# B&R Automation Studio project reAM250plc (part 8)

#### CustomStatemachineRecoater.cpp
```cpp
/*++

Copyright (C) 2024 Institute for Machine Tools and Industrial Management
TUM School of Engineering and Design
Technical University of Munich

All rights reserved.

Redistribution and use in source and binary forms, with or without
modification, are permitted provided that the following conditions are met:
	* Redistributions of source code must retain the above copyright
	  notice, this list of conditions and the following disclaimer.
	* Redistributions in binary form must reproduce the above copyright
	  notice, this list of conditions and the following disclaimer in the
	  documentation and/or other materials provided with the distribution.
	* Neither the name of the Technical University of Munich nor the
	  names of its contributors may be used to endorse or promote products
	  derived from this software without specific prior written permission.

THIS SOFTWARE IS PROVIDED BY THE COPYRIGHT HOLDERS AND CONTRIBUTORS "AS IS" AND
ANY EXPRESS OR IMPLIED WARRANTIES, INCLUDING, BUT NOT LIMITED TO, THE IMPLIED
WARRANTIES OF MERCHANTABILITY AND FITNESS FOR A PARTICULAR PURPOSE ARE
DISCLAIMED. IN NO EVENT SHALL TECHNICAL UNIVERSITY OF MUNICH BE LIABLE FOR ANY
DIRECT, INDIRECT, INCIDENTAL, SPECIAL, EXEMPLARY, OR CONSEQUENTIAL DAMAGES
(INCLUDING, BUT NOT LIMITED TO, PROCUREMENT OF SUBSTITUTE GOODS OR SERVICES;
LOSS OF USE, DATA, OR PROFITS; OR BUSINESS INTERRUPTION) HOWEVER CAUSED AND
ON ANY THEORY OF LIABILITY, WHETHER IN CONTRACT, STRICT LIABILITY, OR TORT
(INCLUDING NEGLIGENCE OR OTHERWISE) ARISING IN ANY WAY OUT OF THE USE OF THIS
SOFTWARE, EVEN IF ADVISED OF THE POSSIBILITY OF SUCH DAMAGE.

*/

#include "Framework/Application.hpp"

#include "CustomConstants.hpp"

//include required hardware modules
#include "Modules/IOModule_X20DO6322.hpp"
#include "Modules/IOModule_X20DI6371.hpp"
#include "Modules/MappMotion_SingleAxis.hpp"
#include "Modules/IOModule_X20SC0842.hpp"

namespace BuRCPP {

	class CStateRecoaterAxes_WaitForInit : public CState {
		public:

		std::string getName ()
		{
			return "wait_for_init";
		}

		void Execute (CEnvironment * pEnvironment)
		{
			pEnvironment->setNextState("wait_for_init");
			// access an IO modules
			ioModuleAccess<CMappMotion_SingleLinearAxis> pRecoaterAxisLinearModule (pEnvironment, "RecoaterLinear");
			ioModuleAccess<CMappMotion_SingleLinearAxis> pRecoaterAxisPowderbeltModule (pEnvironment, "RecoaterAxisPowderbelt");

			// check for PC signals
			auto pSignalInitRecoateraxisPowder = pEnvironment->checkSignal ("initpowderaxis");
			auto pSignalInitRecoateraxisLinear = pEnvironment->checkSignal ("initlinearaxis");

			// get journal variables
			auto bInitRecoateraxisPowder = pEnvironment->getBoolValue(JOURNALVARIABLE_INITRECOATERPOWDERBELT);
			auto bInitRecoateraxisLinear = pEnvironment->getBoolValue(JOURNALVARIABLE_INITRECOATERLINEAR);

			if(bInitRecoateraxisPowder && bInitRecoateraxisLinear)
			{
				// wait for PC signal to init
				pEnvironment->setNextState("init");
			}
			else if(pSignalInitRecoateraxisPowder)
			{
				pEnvironment->setBoolValue(JOURNALVARIABLE_INITRECOATERPOWDERBELT, true);
				pSignalInitRecoateraxisPowder->setBoolResult("success", true);
				pSignalInitRecoateraxisPowder->finishProcessing ();
			}
			else if (pSignalInitRecoateraxisLinear)
			{
				pEnvironment->setBoolValue(JOURNALVARIABLE_INITRECOATERLINEAR, true);
				pSignalInitRecoateraxisLinear->setBoolResult("success", true);
				pSignalInitRecoateraxisLinear->finishProcessing ();
			}
			else if (pRecoaterAxisLinearModule-> isError () || pRecoaterAxisPowderbeltModule-> isError ())
			{
				pEnvironment->setNextState ("error");
			}
			else
			{
				pEnvironment->setNextState("wait_for_init");
			}

		}
	};

	class CStateRecoaterAxes_Init : public CState {
		public:

		std::string getName ()
		{
			return "init";
		}

		void Execute (CEnvironment * pEnvironment)
		{
			// access an IO modules
			ioModuleAccess<CMappMotion_SingleLinearAxis> pRecoaterAxisLinearModule (pEnvironment, "RecoaterLinear");
			ioModuleAccess<CMappMotion_SingleLinearAxis> pRecoaterAxisPowderbeltModule (pEnvironment, "RecoaterAxisPowderbelt");

			if (pRecoaterAxisLinearModule->canSetPower () && pRecoaterAxisPowderbeltModule->canSetPower () )
			{
				if(pRecoaterAxisLinearModule->isReferenced () && pRecoaterAxisLinearModule->isReferenced ())
				{
					pRecoaterAxisLinearModule->setPower(true);
					pRecoaterAxisPowderbeltModule->setPower(true);
					pEnvironment->setNextState ("idle");
				}
				else
				{
					pRecoaterAxisLinearModule->setPowerOnAndStartReference ();
					pRecoaterAxisPowderbeltModule->setPowerOnAndStartReference ();
					pEnvironment->setNextState ("wait_for_referencing");
				}

			}
			else if (pRecoaterAxisLinearModule-> isError () || pRecoaterAxisPowderbeltModule-> isError ())
			{
				pEnvironment->setNextState ("error");
			}
			else
			{
				pEnvironment->setNextState ("init");
			}

		}
	};

	class CStateRecoaterAxes_Idle : public CState {
		public:

		std::string getName ()
		{
			return "idle";
		}

		void Execute (CEnvironment * pEnvironment)
		{
			pEnvironment->setNextState("idle");

			// access an IO modules
			ioModuleAccess<CMappMotion_SingleLinearAxis> pRecoaterAxisLinearModule (pEnvironment, "RecoaterLinear");
			ioModuleAccess<CMappMotion_SingleLinearAxis> pRecoaterAxisPowderbeltModule (pEnvironment, "RecoaterAxisPowderbelt");

			// check for PC signals
			auto pSignalReferenceAxis = pEnvironment->checkSignal ("referenceaxis");
			auto pSignalSingleAxisMovement = pEnvironment->checkSignal ("triggersingleaxismovement");
			auto pSignalDualAxisMovement = pEnvironment->checkSignal ("recoaterdualaxismovement");

			if (pSignalReferenceAxis)
			{
				bool referenceRecoaterAxisLinear = pSignalReferenceAxis->getBoolParameter("reference_recoateraxis_linear");
				bool referenceRecoaterAxisPowder = pSignalReferenceAxis->getBoolParameter("reference_recoateraxis_powder");

				if (referenceRecoaterAxisLinear || referenceRecoaterAxisLinear)
				{
					pEnvironment->setIntegerValue(JOURNALVARIABLE_REFERENCERECOATERPOWDERBELT, referenceRecoaterAxisPowder);
					pEnvironment->setIntegerValue(JOURNALVARIABLE_REFERENCERECOATERLINEAR, referenceRecoaterAxisLinear);
					pEnvironment->setNextState("manual_referencing");
					pSignalReferenceAxis->finishProcessing ();
					return;
				}
			}
			if (pSignalSingleAxisMovement)
			{
				int axisid = pSignalSingleAxisMovement->getInt32Parameter("axisid");
				if (axisid == AXISID_RECOATELINEAR)
				{
					pEnvironment->setNextState("linear_axis_movement");
					pEnvironment->setIntegerValue(JOURNALVARIABLE_RECOATERLINEARMOVEMENTABSOLUTERELATIVE, pSignalSingleAxisMovement->getInt32Parameter("absoluterelative"));
					pEnvironment->setDoubleValue(JOURNALVARIABLE_RECOATERLINEARMOVEMENTPOSITION, pSignalSingleAxisMovement->getInt32Parameter("position") * 0.001);
					pEnvironment->setDoubleValue(JOURNALVARIABLE_RECOATERLINEARMOVEMENTSPEED, pSignalSingleAxisMovement->getInt32Parameter("speed") * 0.001);
					pEnvironment->setDoubleValue(JOURNALVARIABLE_RECOATERLINEARMOVEMENTACCELERATION, pSignalSingleAxisMovement->getInt32Parameter("acceleration") * 0.001);
					pSignalSingleAxisMovement->finishProcessing ();
					return;
				}
				else if (axisid == AXISID_RECOATERPOWDERBELT)
				{
					pEnvironment->setNextState("powder_belt_axis_movement");
					pEnvironment->setIntegerValue(JOURNALVARIABLE_RECOATERPOWDERBELTMOVEMENTABSOLUTERELATIVE, pSignalSingleAxisMovement->getInt32Parameter("absoluterelative"));
					pEnvironment->setDoubleValue(JOURNALVARIABLE_RECOATERPOWDERBELTMOVEMENTPOSITION, pSignalSingleAxisMovement->getInt32Parameter("position") * 0.001);
					pEnvironment->setDoubleValue(JOURNALVARIABLE_RECOATERPOWDERBELTMOVEMENTSPEED, pSignalSingleAxisMovement->getInt32Parameter("speed") * 0.001);
					pEnvironment->setDoubleValue(JOURNALVARIABLE_RECOATERPOWDERBELTMOVEMENTACCELERATION, pSignalSingleAxisMovement->getInt32Parameter("acceleration") * 0.001);
					pSignalSingleAxisMovement->finishProcessing ();
					return;
				}
			}
			if (pSignalDualAxisMovement)
			{
				pEnvironment->setNextState("dual_axis_movement");
				pEnvironment->setDoubleValue(JOURNALVARIABLE_RECOATERMOVEMENTSTARTPOSITION, pSignalDualAxisMovement->getInt32Parameter("recoateraxis_linear_start_position") * 0.001);
				pEnvironment->setDoubleValue(JOURNALVARIABLE_RECOATERMOVEMENTTARGETPOSITION, pSignalDualAxisMovement->getInt32Parameter("recoateraxis_linear_target_position") * 0.001);
				pEnvironment->setDoubleValue(JOURNALVARIABLE_RECOATERMOVEMENTLINEARAXISSPEED, pSignalDualAxisMovement->getInt32Parameter("recoateraxis_linear_speed") * 0.001);
				pEnvironment->setDoubleValue(JOURNALVARIABLE_RECOATERMOVEMENTPOWDERAXISSPEED, pSignalDualAxisMovement->getInt32Parameter("recoateraxis_powder_speed") * 0.001);
				pEnvironment->setDoubleValue(JOURNALVARIABLE_RECOATERMOVEMENTLINEARAXISACCELERATION, pSignalDualAxisMovement->getInt32Parameter("recoater_axes_linear_acceleration") * 0.001);
				pEnvironment->setDoubleValue(JOURNALVARIABLE_RECOATERMOVEMENTPOWDERAXISACCELERATION, pSignalDualAxisMovement->getInt32Parameter("recoater_axes_powder_acceleration") * 0.001);
				pSignalDualAxisMovement->finishProcessing ();
			}
			if (pRecoaterAxisLinearModule-> isError () || pRecoaterAxisPowderbeltModule-> isError ())
			{
				pEnvironment->setNextState ("error");
			}
		}
	};

	class CStateRecoaterAxes_LinearAxisMovement : public CState {
		public:

		std::string getName ()
		{
			return "linear_axis_movement";
		}

		void Execute (CEnvironment * pEnvironment)
		{
			pEnvironment->setNextState("linear_axis_movement");

			// access an IO modules
			ioModuleAccess<CMappMotion_SingleLinearAxis> pRecoaterAxisLinearModule (pEnvironment, "RecoaterLinear");

			if (pRecoaterAxisLinearModule->canMoveAxis ())
			{
				auto absoluterelative = pEnvironment->getInt32Value(JOURNALVARIABLE_RECOATERLINEARMOVEMENTABSOLUTERELATIVE);
				auto position = pEnvironment->getDoubleValue(JOURNALVARIABLE_RECOATERLINEARMOVEMENTPOSITION);
				auto speed = pEnvironment->getDoubleValue(JOURNALVARIABLE_RECOATERLINEARMOVEMENTSPEED);
				auto acceleration = pEnvironment->getDoubleValue(JOURNALVARIABLE_RECOATERLINEARMOVEMENTACCELERATION);

				if (absoluterelative == AXISMOVEMENT_ABSOLUTE){
					pRecoaterAxisLinearModule->moveAxisAbsolute (position, speed, acceleration);

				}else if (absoluterelative == AXISMOVEMENT_RELATIVE){
					pRecoaterAxisLinearModule->moveAxisRelative (position, speed, acceleration);
				}
				pEnvironment->setNextState ("wait_for_linear_axis_movement");
			}
			else if (pRecoaterAxisLinearModule-> isError ())
			{
				pEnvironment->setNextState ("error");
			}
			else
			{
				pEnvironment->setNextState ("linear_axis_movement");
			}
		}

	};

	class CStateRecoaterAxes_WaitForLinearAxisMovement : public CState {
		public:

		std::string getName ()
		{
			return "wait_for_linear_axis_movement";
		}

		void Execute (CEnvironment * pEnvironment)
		{
			pEnvironment->setNextState("wait_for_linear_axis_movement");

			// access an IO modules
			ioModuleAccess<CMappMotion_SingleLinearAxis> pRecoaterAxisLinearModule (pEnvironment, "RecoaterLinear");

			if (pRecoaterAxisLinearModule->isInPosition())
			{
				pEnvironment->setNextState ("idle");
			}
			else if (pRecoaterAxisLinearModule-> isError ())
			{
				pEnvironment->setNextState ("error");
			}
			else
			{
				pEnvironment->setNextState ("wait_for_linear_axis_movement");
			}

		}

	};

	class CStateRecoaterAxes_PowderBeltAxisMovement : public CState {
		public:

		std::string getName ()
		{
			return "powder_belt_axis_movement";
		}

		void Execute (CEnvironment * pEnvironment)
		{
			pEnvironment->setNextState("powder_belt_axis_movement");

			// access an IO modules
			ioModuleAccess<CMappMotion_SingleLinearAxis> pRecoaterAxisPowderbeltModule (pEnvironment, "RecoaterAxisPowderbelt");

			if (pRecoaterAxisPowderbeltModule->canMoveAxis ())
			{
				auto absoluterelative = pEnvironment->getInt32Value(JOURNALVARIABLE_RECOATERPOWDERBELTMOVEMENTABSOLUTERELATIVE);
				auto position = pEnvironment->getDoubleValue(JOURNALVARIABLE_RECOATERPOWDERBELTMOVEMENTPOSITION);
				auto speed = pEnvironment->getDoubleValue(JOURNALVARIABLE_RECOATERPOWDERBELTMOVEMENTSPEED);
				auto acceleration = pEnvironment->getDoubleValue(JOURNALVARIABLE_RECOATERPOWDERBELTMOVEMENTACCELERATION);

				if (absoluterelative == AXISMOVEMENT_ABSOLUTE){
					pRecoaterAxisPowderbeltModule->moveAxisAbsolute (position, speed, acceleration);

				}else if (absoluterelative == AXISMOVEMENT_RELATIVE){
					pRecoaterAxisPowderbeltModule->moveAxisRelative (position, speed, acceleration);
				}
				pEnvironment->setNextState ("wait_for_powder_belt_axis_movement");
			}
			else if (pRecoaterAxisPowderbeltModule-> isError ())
			{
				pEnvironment->setNextState ("error");
			}
			else
			{
				pEnvironment->setNextState ("powder_belt_axis_movement");
			}
		}

	};

	class CStateRecoaterAxes_WaitForPowderBeltAxisMovement : public CState {
		public:

		std::string getName ()
		{
			return "wait_for_powder_belt_axis_movement";
		}

		void Execute (CEnvironment * pEnvironment)
		{
			pEnvironment->setNextState("wait_for_powder_belt_axis_movement");

			// access an IO modules
			ioModuleAccess<CMappMotion_SingleLinearAxis> pRecoaterAxisPowderbeltModule (pEnvironment, "RecoaterAxisPowderbelt");

			if (pRecoaterAxisPowderbeltModule->isInPosition())
			{
				pEnvironment->setNextState ("idle");
			}
			else if (pRecoaterAxisPowderbeltModule-> isError ())
			{
				pEnvironment->setNextState ("error");
			}
			else
			{
				pEnvironment->setNextState ("wait_for_powder_belt_axis_movement");
			}

		}

	};

	class CStateRecoaterAxes_DualAxisMovement : public CState {
		public:

		std::string getName ()
		{
			return "dual_axis_movement";
		}

		void Execute (CEnvironment * pEnvironment)
		{
			pEnvironment->setNextState("dual_axis_movement");

			// access an IO modules
			ioModuleAccess<CMappMotion_SingleLinearAxis> pRecoaterAxisLinearModule (pEnvironment, "RecoaterLinear");
			ioModuleAccess<CMappMotion_SingleLinearAxis> pRecoaterAxisPowderbeltModule (pEnvironment, "RecoaterAxisPowderbelt");

			if (pRecoaterAxisLinearModule->canMoveAxis () && pRecoaterAxisPowderbeltModule->canMoveAxis ())
			{
				auto recoateraxis_linear_start_position = pEnvironment->getDoubleValue(JOURNALVARIABLE_RECOATERMOVEMENTSTARTPOSITION);
				auto recoateraxis_linear_target_position = pEnvironment->getDoubleValue(JOURNALVARIABLE_RECOATERMOVEMENTTARGETPOSITION);
				auto recoateraxis_linear_speed = pEnvironment->getDoubleValue(JOURNALVARIABLE_RECOATERMOVEMENTLINEARAXISSPEED);
				auto recoateraxis_powder_speed = pEnvironment->getDoubleValue(JOURNALVARIABLE_RECOATERMOVEMENTPOWDERAXISSPEED);
				auto recoater_axes_linear_acceleration = pEnvironment->getDoubleValue(JOURNALVARIABLE_RECOATERMOVEMENTLINEARAXISACCELERATION);
				auto recoater_axes_powder_acceleration = pEnvironment->getDoubleValue(JOURNALVARIABLE_RECOATERMOVEMENTPOWDERAXISACCELERATION);

				pRecoaterAxisLinearModule->moveAxisAbsolute (recoateraxis_linear_target_position, recoateraxis_linear_speed, recoater_axes_linear_acceleration);
				auto recoateraxis_powder_target_position = ((-(recoateraxis_linear_target_position-recoateraxis_linear_start_position))/recoateraxis_linear_speed)*recoateraxis_powder_speed;
				pRecoaterAxisPowderbeltModule->moveAxisRelative (recoateraxis_powder_target_position, recoateraxis_powder_speed, recoater_axes_powder_acceleration);

				pEnvironment->setNextState ("wait_for_dual_axis_movement");
			}
			else if (pRecoaterAxisLinearModule-> isError () || pRecoaterAxisPowderbeltModule-> isError ())
			{
				pEnvironment->setNextState ("error");
			}
			else
			{
				pEnvironment->setNextState ("dual_axis_movement");
			}
		}

	};

	class CStateRecoaterAxes_WaitForDualAxisMovement : public CState {
		public:

		std::string getName ()
		{
			return "wait_for_dual_axis_movement";
		}

		void Execute (CEnvironment * pEnvironment)
		{
			pEnvironment->setNextState("wait_for_dual_axis_movement");

			// access an IO modules
			ioModuleAccess<CMappMotion_SingleLinearAxis> pRecoaterAxisLinearModule (pEnvironment, "RecoaterLinear");
			ioModuleAccess<CMappMotion_SingleLinearAxis> pRecoaterAxisPowderbeltModule (pEnvironment, "RecoaterAxisPowderbelt");

			if (pRecoaterAxisLinearModule->isInPosition() && pRecoaterAxisPowderbeltModule->isInPosition())
			{
				pEnvironment->setNextState ("idle");
			}
			else if (pRecoaterAxisLinearModule-> isError () || pRecoaterAxisPowderbeltModule-> isError ())
			{
				pEnvironment->setNextState ("error");
			}
			else
			{
				pEnvironment->setNextState ("wait_for_dual_axis_movement");
			}

		}

	};

	class CStateRecoaterAxes_ManualReferencing : public CState {
		public:

		std::string getName ()
		{
			return "manual_referencing";
		}

		void Execute (CEnvironment * pEnvironment)
		{
			// access an IO modules
			ioModuleAccess<CMappMotion_SingleLinearAxis> pRecoaterAxisLinearModule (pEnvironment, "RecoaterLinear");
			ioModuleAccess<CMappMotion_SingleLinearAxis> pRecoaterAxisPowderbeltModule (pEnvironment, "RecoaterAxisPowderbelt");

			auto referenceRecoaterAxisLinear = pEnvironment->getInt32Value(JOURNALVARIABLE_REFERENCERECOATERLINEAR);
			auto referenceRecoaterAxisPowder = pEnvironment->getInt32Value(JOURNALVARIABLE_REFERENCERECOATERPOWDERBELT);

			if (pRecoaterAxisLinearModule-> isError () || pRecoaterAxisPowderbeltModule-> isError ())
			{
				pEnvironment->setNextState ("error");
			}
			else if (referenceRecoaterAxisLinear || referenceRecoaterAxisPowder)
			{
				if (referenceRecoaterAxisLinear)
				{
					pRecoaterAxisLinearModule->startReference ();
				}
				if (referenceRecoaterAxisPowder)
				{
					pRecoaterAxisPowderbeltModule->startReference ();
				}
				pEnvironment->setNextState("wait_for_referencing");
			}
			else
			{
				pEnvironment->setNextState("manual_referencing");
			}

		}

	};

	class CStateRecoaterAxes_WaitForReferencing : public CState {
		public:

		std::string getName ()
		{
			return "wait_for_referencing";
		}

		void Execute (CEnvironment * pEnvironment)
		{
			pEnvironment->setNextState("wait_for_referencing");

			// access an IO modules
			ioModuleAccess<CMappMotion_SingleLinearAxis> pRecoaterAxisLinearModule (pEnvironment, "RecoaterLinear");
			ioModuleAccess<CMappMotion_SingleLinearAxis> pRecoaterAxisPowderbeltModule (pEnvironment, "RecoaterAxisPowderbelt");

			if (pRecoaterAxisLinearModule-> isError () || pRecoaterAxisPowderbeltModule-> isError ())
			{
				pEnvironment->setNextState ("error");
			}
			else if(pRecoaterAxisLinearModule->isReferenced () && pRecoaterAxisPowderbeltModule->isReferenced ())
			{
				pEnvironment->setNextState("idle");
			}
			else
			{
				pEnvironment->setNextState("wait_for_referencing");
			}

		}

	};

	class CStateRecoaterAxes_Error : public CState {
		public:

		std::string getName ()
		{
			return "error";
		}

		void Execute (CEnvironment * pEnvironment)
		{
			pEnvironment->setNextState("error");

			// access an IO modules
			ioModuleAccess<CMappMotion_SingleLinearAxis> pRecoaterAxisLinearModule (pEnvironment, "RecoaterLinear");
			ioModuleAccess<CMappMotion_SingleLinearAxis> pRecoaterAxisPowderbeltModule (pEnvironment, "RecoaterAxisPowderbelt");
			ioModuleAccess<CIOModule_X20SC0842> pSafeDigitalInputModule115KF53 (pEnvironment, "115KF53"); //acknowledge button

			if(pSafeDigitalInputModule115KF53->getInput(2) == 1) //acknowledge button pressed
			{
				pRecoaterAxisLinearModule->resetError ();
				pRecoaterAxisPowderbeltModule->resetError ();
			}

			if (pRecoaterAxisLinearModule-> isError () || pRecoaterAxisPowderbeltModule-> isError ())
			{
				pEnvironment->setNextState ("error");
			}
			else
			{
				pEnvironment->setNextState ("init");
			}

		}

	};

	class CStateHandlerRecoaterAxes : public CStateHandler {
		public:

		CStateHandlerRecoaterAxes (CApplication* pApplication)
			// retrieve the journal group variable
			: CStateHandler (pApplication->getJournal(), "recoater_axes", pApplication->getModuleHandler (), JOURNALGROUP_RECOATER_AXES)
		{
			// register state machines
			addState (std::make_shared<CStateRecoaterAxes_WaitForInit> ());
			addState (std::make_shared<CStateRecoaterAxes_Init> ());
			addState (std::make_shared<CStateRecoaterAxes_Idle> ());
			addState (std::make_shared<CStateRecoaterAxes_LinearAxisMovement> ());
			addState (std::make_shared<CStateRecoaterAxes_WaitForLinearAxisMovement> ());
			addState (std::make_shared<CStateRecoaterAxes_PowderBeltAxisMovement> ());
			addState (std::make_shared<CStateRecoaterAxes_WaitForPowderBeltAxisMovement> ());
			addState (std::make_shared<CStateRecoaterAxes_DualAxisMovement> ());
			addState (std::make_shared<CStateRecoaterAxes_WaitForDualAxisMovement> ());
			addState (std::make_shared<CStateRecoaterAxes_ManualReferencing> ());
			addState (std::make_shared<CStateRecoaterAxes_WaitForReferencing> ());
			addState (std::make_shared<CStateRecoaterAxes_Error> ());

			// register journal variables
			registerIntegerValue("recoater_powder_absoluterelative", JOURNALVARIABLE_RECOATERPOWDERBELTMOVEMENTABSOLUTERELATIVE, 0, 1);
			registerDoubleValue("recoater_powder_position", JOURNALVARIABLE_RECOATERPOWDERBELTMOVEMENTPOSITION, -1000.0, 1000.0, 20000000);
			registerDoubleValue("recoater_powder_speed", JOURNALVARIABLE_RECOATERPOWDERBELTMOVEMENTSPEED, 0.0, 1000.0, 20000000);
			registerDoubleValue("recoater_powder_acceleration", JOURNALVARIABLE_RECOATERPOWDERBELTMOVEMENTACCELERATION, 0.0, 1000.0, 20000000);
			registerIntegerValue("recoater_powder_referencing", JOURNALVARIABLE_REFERENCERECOATERPOWDERBELT, 0, 1);
			registerIntegerValue("Recoaterlinear_absoluterelative", JOURNALVARIABLE_RECOATERLINEARMOVEMENTABSOLUTERELATIVE, 0, 1);
			registerDoubleValue("recoaterlinear_position", JOURNALVARIABLE_RECOATERLINEARMOVEMENTPOSITION, -1000.0, 1000.0, 20000000);
			registerDoubleValue("recoaterlinear_speed", JOURNALVARIABLE_RECOATERLINEARMOVEMENTSPEED, 0.0, 1000.0, 20000000);
			registerDoubleValue("recoaterlinear_acceleration", JOURNALVARIABLE_RECOATERLINEARMOVEMENTACCELERATION, 0.0, 1000.0, 20000000);
			registerIntegerValue("recoaterlinear_referencing", JOURNALVARIABLE_REFERENCERECOATERLINEAR, 0, 1);

			registerDoubleValue("recoating_startposition", JOURNALVARIABLE_RECOATERMOVEMENTSTARTPOSITION, -1000.0, 1000.0, 20000000);
			registerDoubleValue("recoating_targetposition", JOURNALVARIABLE_RECOATERMOVEMENTTARGETPOSITION, -1000.0, 1000.0, 20000000);
			registerDoubleValue("recoating_linearaxisspeed", JOURNALVARIABLE_RECOATERMOVEMENTLINEARAXISSPEED, -1000.0, 1000.0, 20000000);
			registerDoubleValue("recoating_powderaxisspeed", JOURNALVARIABLE_RECOATERMOVEMENTPOWDERAXISSPEED, -1000.0, 1000.0, 20000000);
			registerDoubleValue("recoating_linearaxisacceleration", JOURNALVARIABLE_RECOATERMOVEMENTLINEARAXISACCELERATION, -1000.0, 1000.0, 20000000);
			registerDoubleValue("recoating_powderaxisacceleration", JOURNALVARIABLE_RECOATERMOVEMENTPOWDERAXISACCELERATION, -1000.0, 1000.0, 20000000);

			registerBoolValue("init_powderaxis", JOURNALVARIABLE_INITRECOATERPOWDERBELT);
			registerBoolValue("init_linearaxis", JOURNALVARIABLE_INITRECOATERLINEAR);

			// register signals
			auto pSignalInitRecoateraxisPowder = registerSignal ("initpowderaxis", 4, 1000);
			pSignalInitRecoateraxisPowder->addBoolResult ("success", false);

			auto pSignalInitRecoateraxisLinear = registerSignal ("initlinearaxis", 4, 1000);
			pSignalInitRecoateraxisLinear->addBoolResult ("success", false);

			auto pSignalSingleAxisMovement = registerSignal ("triggersingleaxismovement", 4, 1000);
			pSignalSingleAxisMovement->addInt32Parameter ("axisid", 0);
			pSignalSingleAxisMovement->addInt32Parameter ("absoluterelative", 0);
			pSignalSingleAxisMovement->addInt32Parameter ("position", 0);
			pSignalSingleAxisMovement->addInt32Parameter ("speed", 0);
			pSignalSingleAxisMovement->addInt32Parameter ("acceleration", 0);
			pSignalSingleAxisMovement->addBoolResult ("success", false);

			auto pSignalReferenceAxis = registerSignal ("referenceaxis", 4, 1000);
			pSignalReferenceAxis->addBoolParameter ("reference_platform", false);
			pSignalReferenceAxis->addBoolParameter ("reference_powderreservoir", false);
			pSignalReferenceAxis->addBoolParameter ("reference_recoateraxis_powder", false);
			pSignalReferenceAxis->addBoolParameter ("reference_recoateraxis_linear", false);
			pSignalReferenceAxis->addBoolResult ("success", false);

			auto pSignalRecoaterDualAxisMovement = registerSignal ("recoaterdualaxismovement", 4, 1000);
			pSignalRecoaterDualAxisMovement->addInt32Parameter ("recoateraxis_linear_start_position", 0);
			pSignalRecoaterDualAxisMovement->addInt32Parameter ("recoateraxis_linear_target_position", 0);
			pSignalRecoaterDualAxisMovement->addInt32Parameter ("recoateraxis_linear_speed", 0);
			pSignalRecoaterDualAxisMovement->addInt32Parameter ("recoateraxis_powder_speed", 0);
			pSignalRecoaterDualAxisMovement->addInt32Parameter ("recoater_axes_linear_acceleration", 0);
			pSignalRecoaterDualAxisMovement->addInt32Parameter ("recoater_axes_powder_acceleration", 0);
			pSignalRecoaterDualAxisMovement->addBoolResult ("success", false);

		}

		virtual ~CStateHandlerRecoaterAxes ()
		{
		}

	};

	void registerRecoaterAxesStateHandler (CApplication * pApplication)
	{
		auto pRecoaterAxesStateHandler = std::make_shared<CStateHandlerRecoaterAxes> (pApplication);
		//pMainStateHandler->setCycleTime (20);
		pRecoaterAxesStateHandler->setDebugVariables (CURRENT_STATE_RECOATER_AXES, 80);
		pApplication->registerStateHandler (pRecoaterAxesStateHandler);
	}

}
```

#### CustomStatemachineO2Sensor.cpp
```cpp
/*++

Copyright (C) 2024 Institute for Machine Tools and Industrial Management
TUM School of Engineering and Design
Technical University of Munich

All rights reserved.

Redistribution and use in source and binary forms, with or without
modification, are permitted provided that the following conditions are met:
	* Redistributions of source code must retain the above copyright
	  notice, this list of conditions and the following disclaimer.
	* Redistributions in binary form must reproduce the above copyright
	  notice, this list of conditions and the following disclaimer in the
	  documentation and/or other materials provided with the distribution.
	* Neither the name of the Technical University of Munich nor the
	  names of its contributors may be used to endorse or promote products
	  derived from this software without specific prior written permission.

THIS SOFTWARE IS PROVIDED BY THE COPYRIGHT HOLDERS AND CONTRIBUTORS "AS IS" AND
ANY EXPRESS OR IMPLIED WARRANTIES, INCLUDING, BUT NOT LIMITED TO, THE IMPLIED
WARRANTIES OF MERCHANTABILITY AND FITNESS FOR A PARTICULAR PURPOSE ARE
DISCLAIMED. IN NO EVENT SHALL TECHNICAL UNIVERSITY OF MUNICH BE LIABLE FOR ANY
DIRECT, INDIRECT, INCIDENTAL, SPECIAL, EXEMPLARY, OR CONSEQUENTIAL DAMAGES
(INCLUDING, BUT NOT LIMITED TO, PROCUREMENT OF SUBSTITUTE GOODS OR SERVICES;
LOSS OF USE, DATA, OR PROFITS; OR BUSINESS INTERRUPTION) HOWEVER CAUSED AND
ON ANY THEORY OF LIABILITY, WHETHER IN CONTRACT, STRICT LIABILITY, OR TORT
(INCLUDING NEGLIGENCE OR OTHERWISE) ARISING IN ANY WAY OUT OF THE USE OF THIS
SOFTWARE, EVEN IF ADVISED OF THE POSSIBILITY OF SUCH DAMAGE.

*/

#include "Framework/Application.hpp"

#include "CustomConstants.hpp"

//include required hardware modules
#include "Modules/IOModule_X20AI4622.hpp"
#include "Modules/IOModule_X20DO6322.hpp"

namespace BuRCPP {

	class CStateO2Sensor_Init : public CState {
		public:

		std::string getName ()
		{
			return "init";
		}

		void Execute (CEnvironment * pEnvironment)
		{

			// access io modules
			ioModuleAccess<CIOModule_X20AI4622>pAnalogInputModule(pEnvironment, "112KF14"); // oxygen content value module
			ioModuleAccess<CIOModule_X20DO6322> pDigitalOutputModule (pEnvironment, "114KF24"); // measuring range switch

			pDigitalOutputModule->setOutput(6, false); // set measuring range 0 to 25 %

			if (pAnalogInputModule->getIOStatus(1) == 0 && pAnalogInputModule->getIOStatus(2) == 0) { // transitioning to measuring_range_0_to_25_percent
				pEnvironment->setNextState ("measuring_range_0_to_25_percent");
			}
			else {
				pEnvironment->setNextState ("error");
			}
		}
	};

	class CStateO2Sensor_measuring_range_0_to_25_percent : public CState {
		public:

		std::string getName()
		{
			return "measuring_range_0_to_25_percent";
		}

		void Execute(CEnvironment* pEnvironment)
		{
			// access io modules
			ioModuleAccess<CIOModule_X20AI4622>pAnalogInputModule(pEnvironment, "112KF14"); // oxygen content value module
			ioModuleAccess<CIOModule_X20DO6322> pDigitalOutputModule(pEnvironment, "114KF24"); // measuring range switch

			// Signal from PC
			auto pSignalSensorTest = pEnvironment->checkSignal ("sensortest");

			double o2inpercent_chamber = (pAnalogInputModule->getInputCurrentInAmpere(2)-0.004)*((O2SENSORCHAMBER_RANGE_COARSE_UPPER_INPERCENT-O2SENSORCHAMBER_RANGE_COARSE_LOWER_INPERCENT)/0.016)+O2SENSORCHAMBER_RANGE_COARSE_LOWER_INPERCENT;
			double o2inpercent_filter = (pAnalogInputModule->getInputCurrentInAmpere(1)-0.004)*((O2SENSORFILTER_RANGE_UPPER_INPERCENT-O2SENSORFILTER_RANGE_LOWER_INPERCENT)/0.016)+O2SENSORFILTER_RANGE_LOWER_INPERCENT;

			pEnvironment->setIntegerValue(JOURNALVARIABLE_O2INPPM_CHAMBER, o2inpercent_chamber*10000.0);
			pEnvironment->setIntegerValue(JOURNALVARIABLE_O2INPPM_FILTER, o2inpercent_filter*10000.0);

			if (o2inpercent_chamber*10000 >= O2SENSORCHAMBER_RANGE_FINE_LOWER_INPPM) {		// oxygen content value >=  1000 ppm
				pDigitalOutputModule->setOutput(6, false);
				pEnvironment->setNextState("measuring_range_0_to_25_percent");
			}
			else {      // oxygen content value < 1000 ppm
				pDigitalOutputModule->setOutput(6, true);
				pEnvironment->setNextState("measuring_range_0_to_1000ppm");
			}
			if (pSignalSensorTest) { // Signal from PC
				pEnvironment->setNextState("sensor_test");
				pSignalSensorTest->finishProcessing ();
			}
			if (pAnalogInputModule->getIOStatus(1) != 0 && pAnalogInputModule->getIOStatus(2) != 0) { // transitioning to error
				pEnvironment->setNextState ("error");
			}

		}

	};

	class CStateO2Sensor_measuring_range_0_to_1000ppm : public CState {
		public:

		std::string getName()
		{
			return "measuring_range_0_to_1000ppm";
		}

		void Execute(CEnvironment* pEnvironment)
		{
			// access io modules
			ioModuleAccess<CIOModule_X20AI4622>pAnalogInputModule(pEnvironment, "112KF14"); // oxygen content value module
			ioModuleAccess<CIOModule_X20DO6322> pDigitalOutputModule(pEnvironment, "114KF24"); // measuring range switch

			// Signal from PC

			auto pSignalSensorTest = pEnvironment->checkSignal ("sensortest");

			double o2inppm_chamber = (pAnalogInputModule->getInputCurrentInAmpere(2)-0.004)*((O2SENSORCHAMBER_RANGE_FINE_UPPER_INPPM-O2SENSORCHAMBER_RANGE_FINE_LOWER_INPPM)/0.016)+O2SENSORCHAMBER_RANGE_FINE_LOWER_INPPM;
			double o2inpercent_filter = (pAnalogInputModule->getInputCurrentInAmpere(1)-0.004)*((O2SENSORFILTER_RANGE_UPPER_INPERCENT-O2SENSORFILTER_RANGE_LOWER_INPERCENT)/0.016)+O2SENSORFILTER_RANGE_LOWER_INPERCENT;

			pEnvironment->setIntegerValue(JOURNALVARIABLE_O2INPPM_CHAMBER, o2inppm_chamber);
			pEnvironment->setIntegerValue(JOURNALVARIABLE_O2INPPM_FILTER, o2inpercent_filter*10000.0);

			if (o2inppm_chamber >= O2SENSORCHAMBER_RANGE_FINE_LOWER_INPPM) {// oxygen content value >= 1000 ppm
				pDigitalOutputModule->setOutput(6, false);
				pEnvironment->setNextState("measuring_range_0_to_25_percent");
			}
			else {      // oxygen content value < 1000 ppm
				pDigitalOutputModule->setOutput(6, true);
				pEnvironment->setNextState("measuring_range_0_to_1000ppm");
			}
			if (pSignalSensorTest) { // Signal from PC
				pEnvironment->setNextState("sensor_test");
				pSignalSensorTest->finishProcessing ();
			}
			if (pAnalogInputModule->getIOStatus(1) != 0 && pAnalogInputModule->getIOStatus(2) != 0) { // transitioning to error
				pEnvironment->setNextState ("error");
			}

		}

	};

	class CStateO2Sensor_sensor_test : public CState {
		public:

		std::string getName()
		{
			return "sensor_test";
		}

		void Execute(CEnvironment* pEnvironment)
		{
			// access io modules
			ioModuleAccess<CIOModule_X20DO6322> pDigitalOutputModule(pEnvironment, "114KF24"); // measuring range switch
			ioModuleAccess<CIOModule_X20AI4622>pAnalogInputModule(pEnvironment, "112KF14"); // oxygen content value module

			if (false) {
				pEnvironment->setNextState("sensor_test");
			}
			else {		// transitioning to init
				pEnvironment->setNextState("init");
			}
			if (pAnalogInputModule->getIOStatus(1) != 0 && pAnalogInputModule->getIOStatus(2) != 0) { // transitioning to error
				pEnvironment->setNextState ("error");
			}
		}

	};

	class CStateO2Sensor_error : public CState {
		public:

		std::string getName()
		{
			return "error";
		}

		void Execute(CEnvironment* pEnvironment)
		{
			// access io modules
			ioModuleAccess<CIOModule_X20AI4622>pAnalogInputModule(pEnvironment, "112KF14"); // oxygen content value module

			if (pAnalogInputModule->getIOStatus(1) == 0 && pAnalogInputModule->getIOStatus(2) == 0) { // transitioning to init
				pEnvironment->setNextState ("init");
			}
			else {
				pEnvironment->setNextState ("error");
			}
		}

	};

	class CO2SensorStateHandler : public CStateHandler {
		public:

		CO2SensorStateHandler (CApplication* pApplication)
			// retrieve the journal group variable for this O2Sensor state machine
			: CStateHandler (pApplication->getJournal (), "O2Sensor", pApplication->getModuleHandler (), JOURNALGROUP_O2SENSOR)
		{
			// register all states of this state machine here
			addState (std::make_shared<CStateO2Sensor_Init> ());
			addState (std::make_shared<CStateO2Sensor_measuring_range_0_to_25_percent> ());
			addState(std::make_shared<CStateO2Sensor_measuring_range_0_to_1000ppm>());
			addState(std::make_shared<CStateO2Sensor_sensor_test>());
			addState(std::make_shared<CStateO2Sensor_error>());

			//register signal
			auto pSignalSensorTest = registerSignal ("sensortest", 4, 1000);
			pSignalSensorTest->addBoolResult ("success", false);

			// register journal variables
			registerIntegerValue("o2chamberinppm", JOURNALVARIABLE_O2INPPM_CHAMBER, 0, 250000);
			registerIntegerValue("o2filterinppm", JOURNALVARIABLE_O2INPPM_FILTER, 0, 250000);

		}

		virtual ~CO2SensorStateHandler ()
		{
		}

	};

	void registerO2SensorStateHandler (CApplication * pApplication)
	{
		auto pO2SensorStateHandler = std::make_shared<CO2SensorStateHandler> (pApplication);
		//pMainStateHandler->setCycleTime (20);
		pO2SensorStateHandler->setDebugVariables (CURRENT_STATE_O2SENSOR, 80);
		pApplication->registerStateHandler (pO2SensorStateHandler);
	}

}
```

#### CustomStatemachineGasCirculation.cpp
```cpp
/*++

Copyright (C) 2024 Institute for Machine Tools and Industrial Management
TUM School of Engineering and Design
Technical University of Munich

All rights reserved.

Redistribution and use in source and binary forms, with or without
modification, are permitted provided that the following conditions are met:
	* Redistributions of source code must retain the above copyright
	  notice, this list of conditions and the following disclaimer.
	* Redistributions in binary form must reproduce the above copyright
	  notice, this list of conditions and the following disclaimer in the
	  documentation and/or other materials provided with the distribution.
	* Neither the name of the Technical University of Munich nor the
	  names of its contributors may be used to endorse or promote products
	  derived from this software without specific prior written permission.

THIS SOFTWARE IS PROVIDED BY THE COPYRIGHT HOLDERS AND CONTRIBUTORS "AS IS" AND
ANY EXPRESS OR IMPLIED WARRANTIES, INCLUDING, BUT NOT LIMITED TO, THE IMPLIED
WARRANTIES OF MERCHANTABILITY AND FITNESS FOR A PARTICULAR PURPOSE ARE
DISCLAIMED. IN NO EVENT SHALL TECHNICAL UNIVERSITY OF MUNICH BE LIABLE FOR ANY
DIRECT, INDIRECT, INCIDENTAL, SPECIAL, EXEMPLARY, OR CONSEQUENTIAL DAMAGES
(INCLUDING, BUT NOT LIMITED TO, PROCUREMENT OF SUBSTITUTE GOODS OR SERVICES;
LOSS OF USE, DATA, OR PROFITS; OR BUSINESS INTERRUPTION) HOWEVER CAUSED AND
ON ANY THEORY OF LIABILITY, WHETHER IN CONTRACT, STRICT LIABILITY, OR TORT
(INCLUDING NEGLIGENCE OR OTHERWISE) ARISING IN ANY WAY OUT OF THE USE OF THIS
SOFTWARE, EVEN IF ADVISED OF THE POSSIBILITY OF SUCH DAMAGE.

*/

#include "Framework/Application.hpp"

#include "CustomConstants.hpp"

//include required hardware modules
#include "Modules/IOModule_X20DI6371.hpp"
#include "Modules/IOModule_X20DO6322.hpp"
#include "Modules/IOModule_X20AO4622.hpp"
#include "Modules/IOModule_X20AI4622.hpp"

namespace BuRCPP {
	class CStateGasCirculation_Init : public CState {
		public:

		std::string getName ()
		{
			return "init";
		}

		void Execute (CEnvironment * pEnvironment)
		{
			// access io modules
			ioModuleAccess<CIOModule_X20DO6322> pDigitalOutputModule_1(pEnvironment, "114KF28"); // enable pump
			ioModuleAccess<CIOModule_X20DO6322> pDigitalOutputModule_2(pEnvironment, "114KF25"); // set valves
			ioModuleAccess<CIOModule_X20AO4622> pAnalogOutputModule(pEnvironment, "112KF12"); // setpoint pump
			ioModuleAccess<CIOModule_X20DI6371> pDigitalInputModule_1(pEnvironment, "113KF19");// pump ventilation error
			ioModuleAccess<CIOModule_X20DI6371> pDigitalInputModule_2(pEnvironment, "113KF18");// pump error

			pDigitalOutputModule_1->setOutput(1, false); // disable pump
			pAnalogOutputModule->setOutputVoltageInVolt (1, 0.0); // set setpoint to 0.0 V

			pDigitalOutputModule_2->setOutput(1, false); // close circulation valves
			pDigitalOutputModule_2->setOutput(2, false);

			// Signal from PC
			auto pSignalInitAtmosphereControl = pEnvironment->checkSignal ("initatmospherecontrol");

			if (pSignalInitAtmosphereControl)
			{
				int circulation_on_threshold = pSignalInitAtmosphereControl->getInt32Parameter("o2thresholdcirculationoninppm");
				int circulation_off_threshold = pSignalInitAtmosphereControl->getInt32Parameter("o2thresholdcirculationoffinppm");
				pEnvironment->setIntegerValue(JOURNALVARIABLE_O2_THRESHOLD_CIRCULATION_ON_IN_PPM, circulation_on_threshold);
				pEnvironment->setIntegerValue(JOURNALVARIABLE_O2_THRESHOLD_CIRCULATION_OFF_IN_PPM, circulation_off_threshold);
				pEnvironment->setNextState("idle");
				pSignalInitAtmosphereControl->finishProcessing ();
			}
			else
			{
				pEnvironment->setNextState("init");
			}

			if (pDigitalInputModule_1->getInput(3)==1 || pDigitalInputModule_2->getInput(3)==0)
			{
				pEnvironment->setNextState("error");
			}
		}
	};

class CStateGasCirculation_error : public CState {
	public:

	std::string getName ()
	{
		return "error";
	}

	void Execute (CEnvironment * pEnvironment)
	{
		// access io modules
		ioModuleAccess<CIOModule_X20DI6371> pDigitalInputModule_1(pEnvironment, "113KF19");// pump ventilation error
		ioModuleAccess<CIOModule_X20DI6371> pDigitalInputModule_2(pEnvironment, "113KF18");// pump error

		if (pDigitalInputModule_1->getInput(3)==1 || pDigitalInputModule_2->getInput(3)==0)
		{
			pEnvironment->setNextState("error");
		}
		else
		{
			pEnvironment->setNextState("init");
		}
	}

};

class CStateGasCirculation_idle : public CState {
	public:

	std::string getName ()
	{
		return "idle";
	}

	void Execute (CEnvironment * pEnvironment)
	{
		// access io modules
		ioModuleAccess<CIOModule_X20DI6371> pDigitalInputModule_1(pEnvironment, "113KF19");// pump ventilation error
		ioModuleAccess<CIOModule_X20DI6371> pDigitalInputModule_2(pEnvironment, "113KF18");// pump error
		ioModuleAccess<CIOModule_X20DI6371> pDigitalInputModule_3(pEnvironment, "113KF17");// get circulation valves status
		ioModuleAccess<CIOModule_X20DI6371> pDigitalInputModule_4(pEnvironment, "113KF21");// get vacuum valves status
		ioModuleAccess<CIOModule_X20AO4622> pAnalogOutputModule(pEnvironment, "112KF12"); // setpoint pump
		ioModuleAccess<CIOModule_X20DO6322> pDigitalOutputModule(pEnvironment, "114KF25"); // set valves

		// Signal from PC
		auto pSignalStartGasFlow = pEnvironment->checkSignal ("startgasflow");
		auto pSignalUpdateGasFlowSetpoint = pEnvironment->checkSignal ("updategasflowsetpoint");
		auto pSignalToggleValves = pEnvironment->checkSignal ("togglevalves");

		if (pSignalToggleValves) // toggle gas flow valves
		{
			bool toggle_heat_exchanger_gas_flow_circuit_valve = pSignalToggleValves->getBoolParameter("toggle_lower_gas_flow_circuit_valve");
			bool toggle_chamber_gas_flow_circuit_valve = pSignalToggleValves->getBoolParameter("toggle_upper_gas_flow_circuit_valve");

			pDigitalOutputModule->setOutput(1, toggle_chamber_gas_flow_circuit_valve);
			pDigitalOutputModule->setOutput(2, toggle_heat_exchanger_gas_flow_circuit_valve);

			pSignalToggleValves->finishProcessing ();
		}

		if (pSignalUpdateGasFlowSetpoint)
		{
			int setpointinpercent = pSignalUpdateGasFlowSetpoint->getInt32Parameter("setpointinpercent");
			pEnvironment->setIntegerValue(JOURNALVARIABLE_PUMPSETPOINTINPERCENT, setpointinpercent); //set journalvariable for setpoint
			pSignalUpdateGasFlowSetpoint->finishProcessing ();
		}

		if (pSignalStartGasFlow && pDigitalInputModule_3->getInput(1)==1 && pDigitalInputModule_3->getInput(3)==1 && pDigitalInputModule_4->getInput(2)==1 && pDigitalInputModule_4->getInput(4)==1)
		{
			int setpointinpercent = pSignalStartGasFlow->getInt32Parameter("setpointinpercent");
			pEnvironment->setIntegerValue(JOURNALVARIABLE_PUMPSETPOINTINPERCENT, setpointinpercent); //set journalvariable for setpoint
			pEnvironment->setNextState("wait_for_oxygenlevel");
			pSignalStartGasFlow->finishProcessing ();
		}
		else
		{
			pEnvironment->setNextState("idle");
		}

		if (pDigitalInputModule_1->getInput(3)==1 || pDigitalInputModule_2->getInput(3)==0)
		{
			pEnvironment->setNextState("error");
		}
	}

};

class CStateGasCirculation_wait_for_oxygenlevel : public CState {
	public:

	std::string getName ()
	{
		return "wait_for_oxygenlevel";
	}

	void Execute (CEnvironment * pEnvironment)
	{
		// access io modules
		ioModuleAccess<CIOModule_X20DI6371> pDigitalInputModule_1(pEnvironment, "113KF19"); //pump ventilation error
		ioModuleAccess<CIOModule_X20DI6371> pDigitalInputModule_2(pEnvironment, "113KF18"); //pump error
		ioModuleAccess<CIOModule_X20AI4622>pAnalogInputModule(pEnvironment, "112KF14"); // oxygen content value module

		// Signal from PC
		auto pSignalTurnOffGasFlow = pEnvironment->checkSignal ("turnoffgasflow");
		auto pSignalUpdateGasFlowSetpoint = pEnvironment->checkSignal ("updategasflowsetpoint");

		if (pSignalUpdateGasFlowSetpoint)
		{
			int setpointinpercent = pSignalUpdateGasFlowSetpoint->getInt32Parameter("setpointinpercent");
			pEnvironment->setIntegerValue(JOURNALVARIABLE_PUMPSETPOINTINPERCENT, setpointinpercent); //set journalvariable for setpoint
			pSignalUpdateGasFlowSetpoint->finishProcessing ();
		}

		double o2inpercent_filter = (pAnalogInputModule->getInputCurrentInAmpere(1)-0.004)*((O2SENSORFILTER_RANGE_UPPER_INPERCENT-O2SENSORFILTER_RANGE_LOWER_INPERCENT)/0.016)+O2SENSORFILTER_RANGE_LOWER_INPERCENT;;
		auto circulation_on_o2thresholdinppm = pEnvironment->getInt32Value(JOURNALVARIABLE_O2_THRESHOLD_CIRCULATION_ON_IN_PPM);

		if (o2inpercent_filter*FACTOR_PERCENT_TO_PPM < circulation_on_o2thresholdinppm)
		{
			pEnvironment->setNextState("gas_flow_on");
		}
		else
		{
			pEnvironment->setNextState("wait_for_oxygenlevel");
		}

		if (pSignalTurnOffGasFlow)
		{
			pEnvironment->setNextState("idle");
			pSignalTurnOffGasFlow->finishProcessing ();
		}

		if (pDigitalInputModule_1->getInput(3)==1 || pDigitalInputModule_2->getInput(3)==0)
		{
			pEnvironment->setNextState("error");
		}
	}

};

class CStateGasCirculation_gas_flow_on : public CState {
	public:

	std::string getName ()
	{
		return "gas_flow_on";
	}

	void Execute (CEnvironment * pEnvironment)
	{
		// access io modules
		ioModuleAccess<CIOModule_X20DI6371> pDigitalInputModule_1(pEnvironment, "113KF19");// pump ventilation error
		ioModuleAccess<CIOModule_X20DI6371> pDigitalInputModule_2(pEnvironment, "113KF18");// pump error
		ioModuleAccess<CIOModule_X20DI6371> pDigitalInputModule_3(pEnvironment, "113KF17"); //feedback from circulation valves
		ioModuleAccess<CIOModule_X20DO6322> pDigitalOutputModule_1(pEnvironment, "114KF28"); // enable pump
		ioModuleAccess<CIOModule_X20DO6322> pDigitalOutputModule_2(pEnvironment, "114KF25"); //output vacuum valves
		ioModuleAccess<CIOModule_X20AO4622> pAnalogOutputModule(pEnvironment, "112KF12"); // setpoint pump
		ioModuleAccess<CIOModule_X20AI4622>pAnalogInputModule(pEnvironment, "112KF14"); // oxygen content value module

		// Signal from PC
		auto pSignalTurnOffGasFlow = pEnvironment->checkSignal ("turnoffgasflow");
		auto pSignalUpdateGasFlowSetpoint = pEnvironment->checkSignal ("updategasflowsetpoint");

		if (pSignalUpdateGasFlowSetpoint)
		{
			int setpointinpercent = pSignalUpdateGasFlowSetpoint->getInt32Parameter("setpointinpercent");
			pEnvironment->setIntegerValue(JOURNALVARIABLE_PUMPSETPOINTINPERCENT, setpointinpercent); //set journalvariable for setpoint
			pSignalUpdateGasFlowSetpoint->finishProcessing ();
		}

		pDigitalOutputModule_1->setOutput(1, true); // enable pump
		auto setpointinpercent = pEnvironment->getInt32Value(JOURNALVARIABLE_PUMPSETPOINTINPERCENT);
		auto setpointinvolt = setpointinpercent/10;
		pAnalogOutputModule->setOutputVoltageInVolt (1, setpointinvolt); // set setpoint in V (0 - 10 V)

		double o2inpercent_filter = (pAnalogInputModule->getInputCurrentInAmpere(1)-0.004)*((O2SENSORFILTER_RANGE_UPPER_INPERCENT-O2SENSORFILTER_RANGE_LOWER_INPERCENT)/0.016)+O2SENSORFILTER_RANGE_LOWER_INPERCENT;;
		auto circulation_off_o2thresholdinppm = pEnvironment->getInt32Value(JOURNALVARIABLE_O2_THRESHOLD_CIRCULATION_OFF_IN_PPM);

		if (o2inpercent_filter*FACTOR_PERCENT_TO_PPM < circulation_off_o2thresholdinppm)
		{
			pEnvironment->setNextState("gas_flow_on");
		}
		else
		{
			pDigitalOutputModule_1->setOutput(1, false); // disable pump
			pAnalogOutputModule->setOutputVoltageInVolt (1, 0.0); // set setpoint to 0.0 V
			pEnvironment->setNextState("wait_for_oxygenlevel");
		}

		if (pSignalTurnOffGasFlow)
		{
			pDigitalOutputModule_1->setOutput(1, false); // disable pump
			pAnalogOutputModule->setOutputVoltageInVolt (1, 0.0); // set setpoint to 0.0 V

			pEnvironment->setNextState("idle");
			pSignalTurnOffGasFlow->finishProcessing ();
		}

		if (pDigitalInputModule_1->getInput(3)==1 || pDigitalInputModule_2->getInput(3)==0 || pDigitalInputModule_3->getInput(1)==0 || pDigitalInputModule_3->getInput(3)==0 || pDigitalOutputModule_2->getOutput(4)==1 || pDigitalOutputModule_2->getOutput(5)==1)
		{
			pDigitalOutputModule_1->setOutput(1, false); // disable pump
			pAnalogOutputModule->setOutputVoltageInVolt (1, 0.0); // set setpoint to 0.0 V

			pEnvironment->setNextState("error");
		}
	}

};

class CStateHandlerGasCirculation : public CStateHandler {
	public:

	CStateHandlerGasCirculation (CApplication* pApplication)
		// retrieve the journal group variable for this template state machine
		: CStateHandler (pApplication->getJournal (), "gascirculation", pApplication->getModuleHandler (), JOURNALGROUP_GAS_CIRCULATION)
	{
		// register all states of this state machine here
		addState (std::make_shared<CStateGasCirculation_Init> ());
		addState (std::make_shared<CStateGasCirculation_idle> ());
		addState (std::make_shared<CStateGasCirculation_wait_for_oxygenlevel> ());
		addState (std::make_shared<CStateGasCirculation_gas_flow_on> ());
		addState (std::make_shared<CStateGasCirculation_error> ());

		//register signal
		auto pSignalInitAtmosphereControl = registerSignal ("initatmospherecontrol", 4, 1000);
		pSignalInitAtmosphereControl->addInt32Parameter ("o2thresholdcirculationoninppm", 0);
		pSignalInitAtmosphereControl->addInt32Parameter ("o2thresholdcirculationoffinppm", 0);
		pSignalInitAtmosphereControl->addBoolResult ("success", false);

		auto pSignalToggleValves = registerSignal ("togglevalves", 4, 1000);
		pSignalToggleValves->addBoolParameter ("toggle_lower_gas_flow_circuit_valve", false);
		pSignalToggleValves->addBoolParameter ("toggle_upper_gas_flow_circuit_valve", false);
		pSignalToggleValves->addBoolParameter ("toggle_shielding_gas_valve", false);
		pSignalToggleValves->addBoolParameter ("toggle_chamber_vacuum_valve", false);
		pSignalToggleValves->addBoolParameter ("toggle_zAxis_vacuum_valve", false);
		pSignalToggleValves->addBoolResult ("success", false);

		auto pSignalStartGasFlow = registerSignal ("startgasflow", 4, 1000);
		pSignalStartGasFlow->addInt32Parameter ("setpointinpercent", 0);
		pSignalStartGasFlow->addBoolResult ("success", false);

		auto pSignalUpdateGasFlowSetpoint = registerSignal ("updategasflowsetpoint", 4, 1000);
		pSignalUpdateGasFlowSetpoint->addInt32Parameter ("setpointinpercent", 0);
		pSignalUpdateGasFlowSetpoint->addBoolResult ("success", false);

		auto pSignalTurnOffGasFlow = registerSignal ("turnoffgasflow", 4, 1000);
		pSignalTurnOffGasFlow->addBoolResult ("success", false);

		// register journal variables
		registerIntegerValue("pumpsetpointinpercent", JOURNALVARIABLE_PUMPSETPOINTINPERCENT, 0, 100);
		registerIntegerValue("o2thresholdcirculationoninppm", JOURNALVARIABLE_O2_THRESHOLD_CIRCULATION_ON_IN_PPM, 0, 250000);
		registerIntegerValue("o2thresholdcirculationoffinppm", JOURNALVARIABLE_O2_THRESHOLD_CIRCULATION_OFF_IN_PPM, 0, 250000);

	}

	virtual ~CStateHandlerGasCirculation ()
	{
	}

};

void registerGasCirculationStateHandler (CApplication * pApplication)
{
	auto pGasCirculationStateHandler = std::make_shared<CStateHandlerGasCirculation> (pApplication);
	//pMainStateHandler->setCycleTime (20);
	pGasCirculationStateHandler->setDebugVariables (CURRENT_STATE_GAS_CIRCULATION, 80);
	pApplication->registerStateHandler (pGasCirculationStateHandler);
}

}
```

#### CustomStatemachineVacuumSystem.cpp
```cpp
/*++

Copyright (C) 2024 Institute for Machine Tools and Industrial Management
TUM School of Engineering and Design
Technical University of Munich

All rights reserved.

Redistribution and use in source and binary forms, with or without
modification, are permitted provided that the following conditions are met:
	* Redistributions of source code must retain the above copyright
	  notice, this list of conditions and the following disclaimer.
	* Redistributions in binary form must reproduce the above copyright
	  notice, this list of conditions and the following disclaimer in the
	  documentation and/or other materials provided with the distribution.
	* Neither the name of the Technical University of Munich nor the
	  names of its contributors may be used to endorse or promote products
	  derived from this software without specific prior written permission.

THIS SOFTWARE IS PROVIDED BY THE COPYRIGHT HOLDERS AND CONTRIBUTORS "AS IS" AND
ANY EXPRESS OR IMPLIED WARRANTIES, INCLUDING, BUT NOT LIMITED TO, THE IMPLIED
WARRANTIES OF MERCHANTABILITY AND FITNESS FOR A PARTICULAR PURPOSE ARE
DISCLAIMED. IN NO EVENT SHALL TECHNICAL UNIVERSITY OF MUNICH BE LIABLE FOR ANY
DIRECT, INDIRECT, INCIDENTAL, SPECIAL, EXEMPLARY, OR CONSEQUENTIAL DAMAGES
(INCLUDING, BUT NOT LIMITED TO, PROCUREMENT OF SUBSTITUTE GOODS OR SERVICES;
LOSS OF USE, DATA, OR PROFITS; OR BUSINESS INTERRUPTION) HOWEVER CAUSED AND
ON ANY THEORY OF LIABILITY, WHETHER IN CONTRACT, STRICT LIABILITY, OR TORT
(INCLUDING NEGLIGENCE OR OTHERWISE) ARISING IN ANY WAY OUT OF THE USE OF THIS
SOFTWARE, EVEN IF ADVISED OF THE POSSIBILITY OF SUCH DAMAGE.

*/

#include <cmath>

#include "Framework/Application.hpp"

#include "CustomConstants.hpp"

//include required hardware modules
#include "Modules/IOModule_X20DO6322.hpp"
#include "Modules/IOModule_X20DI6371.hpp"
#include "Modules/IOModule_X20AI4622.hpp"
#include "Modules/MappMotion_SingleAxis.hpp"

namespace BuRCPP {
	class CStateVacuumSystem_Init : public CState {
		public:

		std::string getName ()
		{
			return "init";
		}

		void Execute (CEnvironment * pEnvironment)
		{
			// access io modules
			ioModuleAccess<CIOModule_X20DO6322> pDigitalOutputModule_1(pEnvironment, "114KF28"); // enable pump
			ioModuleAccess<CIOModule_X20DO6322> pDigitalOutputModule_2(pEnvironment, "114KF25"); // set valves
			ioModuleAccess<CIOModule_X20DI6371> pDigitalInputModule_1(pEnvironment, "113KF19");// pressure measurement error
			ioModuleAccess<CIOModule_X20DI6371> pDigitalInputModule_2(pEnvironment, "113KF18");// pump error

			pDigitalOutputModule_1->setOutput(2, false); // disable pump

			pDigitalOutputModule_2->setOutput(4, false); // close vacuum valves
			pDigitalOutputModule_2->setOutput(5, false);

			// Signal from PC
			auto pSignalInitVacuumSystem = pEnvironment->checkSignal ("initvacuumsystem");

			if (pSignalInitVacuumSystem)
			{
				int pressure_threshold_vacuum_off_in_mbar = pSignalInitVacuumSystem->getInt32Parameter("pressurethresholdvacuumoffinmbar");
				pEnvironment->setIntegerValue(JOURNALVARIABLE_PRESSURE_THRESHOLD_VACUUM_OFF_IN_MBAR, pressure_threshold_vacuum_off_in_mbar);
				pEnvironment->setNextState("idle");
				pSignalInitVacuumSystem->finishProcessing ();
			}
			else
			{
				pEnvironment->setNextState("init");
			}

			if (pDigitalInputModule_1->getInput(2)==0 || pDigitalInputModule_2->getInput(5)==1)
			{
				pEnvironment->setNextState("error");
			}
		}
	};

	class CStateVacuumSystem_idle : public CState {
		public:

		std::string getName ()
		{
			return "idle";
		}

		void Execute (CEnvironment * pEnvironment)
		{
			// access io modules
			ioModuleAccess<CIOModule_X20DI6371> pDigitalInputModule_1(pEnvironment, "113KF19");// pressure measurement error
			ioModuleAccess<CIOModule_X20DI6371> pDigitalInputModule_2(pEnvironment, "113KF18");// pump error
			ioModuleAccess<CIOModule_X20DI6371> pDigitalInputModule_3(pEnvironment, "113KF17");// get circulation valves status
			ioModuleAccess<CIOModule_X20DI6371> pDigitalInputModule_4(pEnvironment, "113KF21");// get vacuum valves status
			ioModuleAccess<CIOModule_X20DO6322> pDigitalOutputModule(pEnvironment, "114KF25"); // set valves

			// Signal from PC
			auto pSignalStartVacuumPump = pEnvironment->checkSignal ("startvacuumpump");
			auto pSignalToggleValves = pEnvironment->checkSignal ("togglevalves");

			if (pSignalToggleValves) // toggle gas flow valves
			{
				bool toggle_zAxis_vacuum_valve = pSignalToggleValves->getBoolParameter("toggle_zAxis_vacuum_valve");
				bool toggle_chamber_vacuum_valve = pSignalToggleValves->getBoolParameter("toggle_chamber_vacuum_valve");

				pDigitalOutputModule->setOutput(5, toggle_zAxis_vacuum_valve);
				pDigitalOutputModule->setOutput(4, toggle_chamber_vacuum_valve);
				pSignalToggleValves->finishProcessing ();
			}

			if (pSignalStartVacuumPump && pDigitalInputModule_3->getInput(2)==1 && pDigitalInputModule_3->getInput(4)==1 && pDigitalInputModule_4->getInput(1)==1 && pDigitalInputModule_4->getInput(3)==1)
			{
				pEnvironment->setNextState("vacuum_pump_on");
				pSignalStartVacuumPump->finishProcessing ();
			}
			else
			{
				pEnvironment->setNextState("idle");
			}

			if (pDigitalInputModule_1->getInput(2)==0 || pDigitalInputModule_2->getInput(5)==1)
			{
				pEnvironment->setNextState("error");
			}
		}

	};

	class CStateVacuumSystem_vacuum_pump_on : public CState {
		public:

		std::string getName ()
		{
			return "vacuum_pump_on";
		}

		void Execute (CEnvironment * pEnvironment)
		{
			// access io modules
			ioModuleAccess<CIOModule_X20DI6371> pDigitalInputModule_1(pEnvironment, "113KF19");// pressure measurement error
			ioModuleAccess<CIOModule_X20DI6371> pDigitalInputModule_2(pEnvironment, "113KF18");// pump error
			ioModuleAccess<CIOModule_X20AI4622> pAnalogInputModule(pEnvironment, "112KF15");// pressure in volt
			ioModuleAccess<CIOModule_X20DO6322> pDigitalOutputModule(pEnvironment, "114KF28");// enable vacuum pump

			// Signal from PC
			auto pSignalTurnOffVacuumPump = pEnvironment->checkSignal ("turnoffvacuumpump");

			double pressure_in_volt = pAnalogInputModule->getInputVoltageInVolt(1);
			int pressure_in_mbar = (int) (std::pow(10 , 0.778*(pressure_in_volt - 6.143))); //characteristic curve of the pressure sensor, type-casting to integer
			pEnvironment->setIntegerValue(JOURNALVARIABLE_PRESSURE_IN_MBAR, pressure_in_mbar);
			auto pressure_threshold_vacuum_off_in_mbar = pEnvironment->getInt32Value(JOURNALVARIABLE_PRESSURE_THRESHOLD_VACUUM_OFF_IN_MBAR);

			pDigitalOutputModule->setOutput(2, true); // enable vacuum pump

			if (pSignalTurnOffVacuumPump || (pressure_in_mbar < pressure_threshold_vacuum_off_in_mbar))
			{
				pDigitalOutputModule->setOutput(2, false); // disable vacuum pump
				pEnvironment->setNextState("idle");
				pSignalTurnOffVacuumPump->finishProcessing ();
			}
			else
			{
				pEnvironment->setNextState("vacuum_pump_on");
			}

			if (pDigitalInputModule_1->getInput(2)==0 || pDigitalInputModule_2->getInput(5)==1)
			{
				pDigitalOutputModule->setOutput(2, false); // disable vacuum pump
				pEnvironment->setNextState("error");
			}
		}

	};

	class CStateVacuumSystem_error : public CState {
		public:

		std::string getName ()
		{
			return "error";
		}

		void Execute (CEnvironment * pEnvironment)
		{
			// access io modules
			ioModuleAccess<CIOModule_X20DI6371> pDigitalInputModule_1(pEnvironment, "113KF19");// pressure measurement error
			ioModuleAccess<CIOModule_X20DI6371> pDigitalInputModule_2(pEnvironment, "113KF18");// pump error

			if (pDigitalInputModule_1->getInput(2)==0 || pDigitalInputModule_2->getInput(5)==1)
			{
				pEnvironment->setNextState("error");
			}
			else
			{
				pEnvironment->setNextState("init");
			}
		}

	};

	class CStateHandlerVacuumSystem : public CStateHandler {
		public:

		CStateHandlerVacuumSystem (CApplication* pApplication)
			// retrieve the journal group variable for this vacuum system state machine
			: CStateHandler (pApplication->getJournal (), "vacuumsystem", pApplication->getModuleHandler (), JOURNALGROUP_VACUUMSYSTEM)
		{
			// register all states of this state machine here
			addState (std::make_shared<CStateVacuumSystem_Init> ());
			addState (std::make_shared<CStateVacuumSystem_idle> ());
			addState (std::make_shared<CStateVacuumSystem_vacuum_pump_on> ());
			addState (std::make_shared<CStateVacuumSystem_error> ());

			//register signal
			auto pSignalInitVacuumSystem = registerSignal ("initvacuumsystem", 4, 1000);
			pSignalInitVacuumSystem->addInt32Parameter ("pressurethresholdvacuumoffinmbar", 0);
			pSignalInitVacuumSystem->addBoolResult ("success", false);

			auto pSignalToggleValves = registerSignal ("togglevalves", 4, 1000);
			pSignalToggleValves->addBoolParameter ("toggle_lower_gas_flow_circuit_valve", false);
			pSignalToggleValves->addBoolParameter ("toggle_upper_gas_flow_circuit_valve", false);
			pSignalToggleValves->addBoolParameter ("toggle_shielding_gas_valve", false);
			pSignalToggleValves->addBoolParameter ("toggle_chamber_vacuum_valve", false);
			pSignalToggleValves->addBoolParameter ("toggle_zAxis_vacuum_valve", false);
			pSignalToggleValves->addBoolResult ("success", false);

			auto pSignalStartVacuumPump = registerSignal ("startvacuumpump", 4, 1000);
			pSignalStartVacuumPump->addBoolResult ("success", false);

			auto pSignalTurnOffVacuumPump = registerSignal ("turnoffvacuumpump", 4, 1000);
			pSignalTurnOffVacuumPump->addBoolResult ("success", false);

			// register journal variables
			registerIntegerValue("pressurethresholdvacuumoffinmbar", JOURNALVARIABLE_PRESSURE_THRESHOLD_VACUUM_OFF_IN_MBAR, 0, 1000);
			registerIntegerValue("pressureinmbar", JOURNALVARIABLE_PRESSURE_IN_MBAR, 0, 1000);

		}

		virtual ~CStateHandlerVacuumSystem ()
		{
		}

	};

	void registerVacuumSystemStateHandler (CApplication * pApplication)
	{
		auto pVacuumSystemStateHandler = std::make_shared<CStateHandlerVacuumSystem> (pApplication);
		//pMainStateHandler->setCycleTime (20);
		pVacuumSystemStateHandler->setDebugVariables (CURRENT_STATE_VACUUMSYSTEM, 80);
		pApplication->registerStateHandler (pVacuumSystemStateHandler);
	}

}
```
